FUNCTION FC_RealFormatter : T_SHORT_STR
VAR_INPUT
	iReal:				REAL;
	iNumberOfDecimals:	INT;
END_VAR

FC_RealFormatter := LREAL_TO_FMTSTR(in := iReal, iPrecision := iNumberOfDecimals, bRound := FALSE);

END_FUNCTION

(* stored: Version 1.1.0.1, ProductVersion 3.1.4026.18
   POU FC_RealFormatter: Id {349ebb16-d1d0-4c85-bb9d-56f369a6edca}, SpecialFunc None *)
